{attribute 'GeneratedUsingTerminal: EL6070-0000-0016'}
{attribute addProperty BoxType "EL6070-0000-0016"}
{attribute addProperty Id "EtcSlaveTerminalBaseInfoDataAT %I*InfoData_32EB74EA10"}
{attribute addProperty CRC "3667650902"}
{attribute addProperty Size "10"}
TYPE EL6070_DA9BE956 EXTENDS EtcSlaveTerminalBase :
STRUCT
	{attribute addProperty Name "InfoData"}
	InfoData : InfoData_32EB74EA;
END_STRUCT
END_TYPE

(* stored: Version 1.2.0.0, ProductVersion 3.1.4024.9
   DUT EL6070_DA9BE956: Id {47a1209f-e9cd-46d7-9da4-c1d660234bf2} *)
